FUNCTION_BLOCK FB_AlpacaGet
VAR_INPUT
END_VAR
VAR_OUTPUT
	bBusy               : BOOL;
	bError              : BOOL;
    eStatusCode         : E_AlpacaStatusCode;
END_VAR
VAR_IN_OUT
    fbClient            : FB_IotHttpClient;
END_VAR
VAR
    sUri                : STRING;
    fbRequest           : FB_IotHttpRequest;
	fbJson              : FB_JsonDomParser;
    nState              : UINT;
	jsonDoc             : SJsonValue;
    jsonVal             : SJsonValue;
	bGetContentResult	: BOOL;
	sContent			: STRING(511);
    tSent               : TIME;
END_VAR

// small state machine:
CASE nState OF 
    0:
        // send the request
        IF fbRequest.SendRequest(
                sUri            := sUri,
                fbClient        := fbClient,
                eRequestType    := ETcIotHttpRequestType.HTTP_GET,
                pContent        := 0,
                nContentSize    := 0, 
                fbHeader        := 0) THEN
            nState      := 1;
            bBusy       := TRUE;
            bError      := FALSE;
            eStatusCode := E_AlpacaStatusCode.OK; 
            tSent       := TIME();
        END_IF
    1:
        // wait for the response
        IF NOT fbRequest.bBusy THEN
            bGetContentResult:= fbRequest.GetContent(
                pContent            := ADR(sContent),
                nContentSize        := SIZEOF(sContent),
                bSetNullTermination := TRUE);
            
			IF fbRequest.nStatusCode >= 200 AND fbRequest.nStatusCode < 300 THEN
				jsonDoc := fbRequest.GetJsonDomContent(fbJson);
				IF jsonDoc <> 0 THEN
                    eStatusCode := E_AlpacaStatusCode.OK; 
					bError:= FALSE;
                ELSE
                    bError := TRUE;
                    eStatusCode := E_AlpacaStatusCode.ERROR_WRONG_RESPONSE_CONTENT; 
				END_IF
            ELSE
                bError := TRUE;
                eStatusCode := E_AlpacaStatusCode.ERROR_WRONG_HTTP_STATUS_CODE; 
			END_IF
                
            nState:= 0;
		    bBusy:= FALSE;
		END_IF
END_CASE

METHOD FB_init : BOOL
VAR_INPUT
	bInitRetains : BOOL; // if TRUE, the retain variables are initialized (warm start / cold start)
	bInCopyCode : BOOL;  // if TRUE, the instance afterwards gets moved into the copy code (online change)
    sDeviceName     : STRING;
    nDeviceNumber   : UINT;
    sVariableName   : STRING;
END_VAR
sUri := F_AlpacaFormatUri(sDeviceName, nDeviceNumber, sVariableName);
END_METHOD

METHOD M_FetchResultBool : BOOL
VAR_INPUT
END_VAR
VAR_IN_OUT
    stData : ST_AlpacaGetBool;
END_VAR
VAR
    nTmpInt : DINT;
END_VAR
IF fbJson.HasMember(jsonDoc, 'Value') THEN
    jsonVal:= fbJson.FindMember(jsonDoc, 'Value');
    IF fbJson.IsBool(jsonVal) THEN
        stData.bValue      := fbJson.GetBool(jsonVal);
        stData.eStatusCode := E_AlpacaStatusCode.OK;
        stData.rAge       := TIME_TO_REAL(TIME() - tSent);
    ELSIF fbJson.IsInt(jsonVal) THEN
        nTmpInt := fbJson.GetInt(jsonVal);
        IF nTmpInt = 0 THEN
            stData.bValue := FALSE;
            stData.eStatusCode := E_AlpacaStatusCode.OK;
            stData.rAge       := TIME_TO_REAL(TIME() - tSent);
        ELSIF nTmpInt = 1 THEN
            stData.bValue := TRUE;
            stData.eStatusCode := E_AlpacaStatusCode.OK;
            stData.rAge       := TIME_TO_REAL(TIME() - tSent);
        ELSE
            stData.bValue      := FALSE;
            stData.eStatusCode := E_AlpacaStatusCode.ERROR_WRONG_CONVERSION;
		END_IF
    ELSE
        stData.bValue      := FALSE;
        stData.eStatusCode := E_AlpacaStatusCode.ERROR_WRONG_CONVERSION;
	END_IF
ELSE
    stData.bValue      := FALSE;
    stData.eStatusCode := E_AlpacaStatusCode.ERROR_WRONG_RESPONSE_MEMBER;
END_IF
END_METHOD

METHOD M_FetchResultCoverState : BOOL
VAR_INPUT
END_VAR
VAR_IN_OUT
    stData : ST_AlpacaGetCoverState;
END_VAR
VAR
    nTmpInt : DINT;
END_VAR
IF fbJson.HasMember(jsonDoc, 'Value') THEN
    jsonVal:= fbJson.FindMember(jsonDoc, 'Value');
    IF fbJson.IsInt(jsonVal) THEN
        stData.nValue       := fbJson.GetInt(jsonVal);
        stData.eValue       := stData.nValue;
        stData.sValue       := TO_STRING(stData.eValue);
        stData.eStatusCode  := E_AlpacaStatusCode.OK;
        stData.rAge         := TIME_TO_REAL(TIME() - tSent);
    ELSE
        stData.eValue       := E_AlpacaCoverState.UNKNOWN;
        stData.nValue       := stData.eValue;
        stData.sValue       := TO_STRING(stData.eValue);
        stData.eStatusCode  := E_AlpacaStatusCode.ERROR_WRONG_CONVERSION;
	END_IF
ELSE
    stData.eValue       := E_AlpacaCoverState.UNKNOWN;
    stData.nValue       := stData.eValue;
    stData.sValue       := TO_STRING(stData.eValue);
    stData.eStatusCode := E_AlpacaStatusCode.ERROR_WRONG_RESPONSE_MEMBER;
END_IF
END_METHOD

METHOD M_FetchResultLreal : LREAL
VAR_INPUT
END_VAR
VAR_IN_OUT
    stData : ST_AlpacaGetLreal;
END_VAR
IF fbJson.HasMember(jsonDoc, 'Value') THEN
    jsonVal:= fbJson.FindMember(jsonDoc, 'Value');
    IF fbJson.IsDouble(jsonVal) THEN
        stData.lrValue      := fbJson.GetDouble(jsonVal);
        stData.eStatusCode  := E_AlpacaStatusCode.OK;
        stData.rAge         := TIME_TO_REAL(TIME() - tSent);
    ELSIF fbJson.IsInt(jsonVal) THEN
        stData.lrValue      := DINT_TO_LREAL(fbJson.GetInt(jsonVal));
        stData.eStatusCode  := E_AlpacaStatusCode.OK;
        stData.rAge         := TIME_TO_REAL(TIME() - tSent);
    ELSE
        stData.lrValue      := 0.0;
        stData.eStatusCode  := E_AlpacaStatusCode.ERROR_WRONG_CONVERSION;
	END_IF
ELSE
    stData.lrValue          := 0.0;
    stData.eStatusCode      := E_AlpacaStatusCode.ERROR_WRONG_RESPONSE_MEMBER;
END_IF
END_METHOD

END_FUNCTION_BLOCK

(* stored: Version 1.1.0.1, ProductVersion 3.1.4024.12
   POU FB_AlpacaGet: Id {e750c028-408f-48d9-9d08-604be5efe10f}, SpecialFunc None
   Method FB_init: Id {06ea3e7b-89dd-45d3-a15c-fd165c58c558}
   Method M_FetchResultBool: Id {5aaed2ba-71d6-44e8-aa2b-2982596597d8}
   Method M_FetchResultCoverState: Id {01cb43d9-33fd-457a-8d74-f9ecf2ae8394}
   Method M_FetchResultLreal: Id {b3fa729c-4e24-4a4a-9889-2ce58bdc11e4} *)
